PROGRAM MAIN
VAR
END_VAR

END_PROGRAM

(* stored: Version 1.1.0.1
   POU MAIN: Id {e915e5ad-315a-4d6b-b35a-010ad56c6955} *)
